// TIA Portal V16 export
// export: Created 2022-11-17T15:49:15.2421619Z, ExportSetting WithDefaults, DisplayName Totally Integrated Automation Portal, DisplayVersion V16 Update 6, DisplayName TIA Portal Version Control Interface, DisplayVersion V16 Update 2, DisplayName TIA Portal Openness, DisplayVersion V16 Update 6, DisplayName SINAMICS Startdrive Advanced, DisplayVersion V16 Update 5, DisplayName SINAMICS Startdrive G130, G150, S120, S150, SINAMICS MV, S210, DisplayVersion V16 Update 5, DisplayName SINAMICS Startdrive G110M, G120, G120C, G120D, G120P, G115D, DisplayVersion V16 Update 5, DisplayName STEP 7 Professional, DisplayVersion V16 Update 6, DisplayName STEP 7 Safety, DisplayVersion V16, DisplayName WinCC Advanced, DisplayVersion V16 Update 6
FUNCTION "FC06_TechnoplatCycle" : Void   // FC6, LAD
TITLE = Machine cycle
{ S7_Optimized_Access := 'FALSE' }
AUTHOR : Robopac
VERSION : 0.0
// stored: AutoNumber false, IsIECCheckEnabled false, SetENOAutomatically false, UDAEnableTagReadback false
   VAR_TEMP   // added for the SCL form of the ladder/FBD networks
      _w1 : Bool;
   END_VAR
BEGIN

REGION Network 1: Machine cycle: M0.0 Start cycle
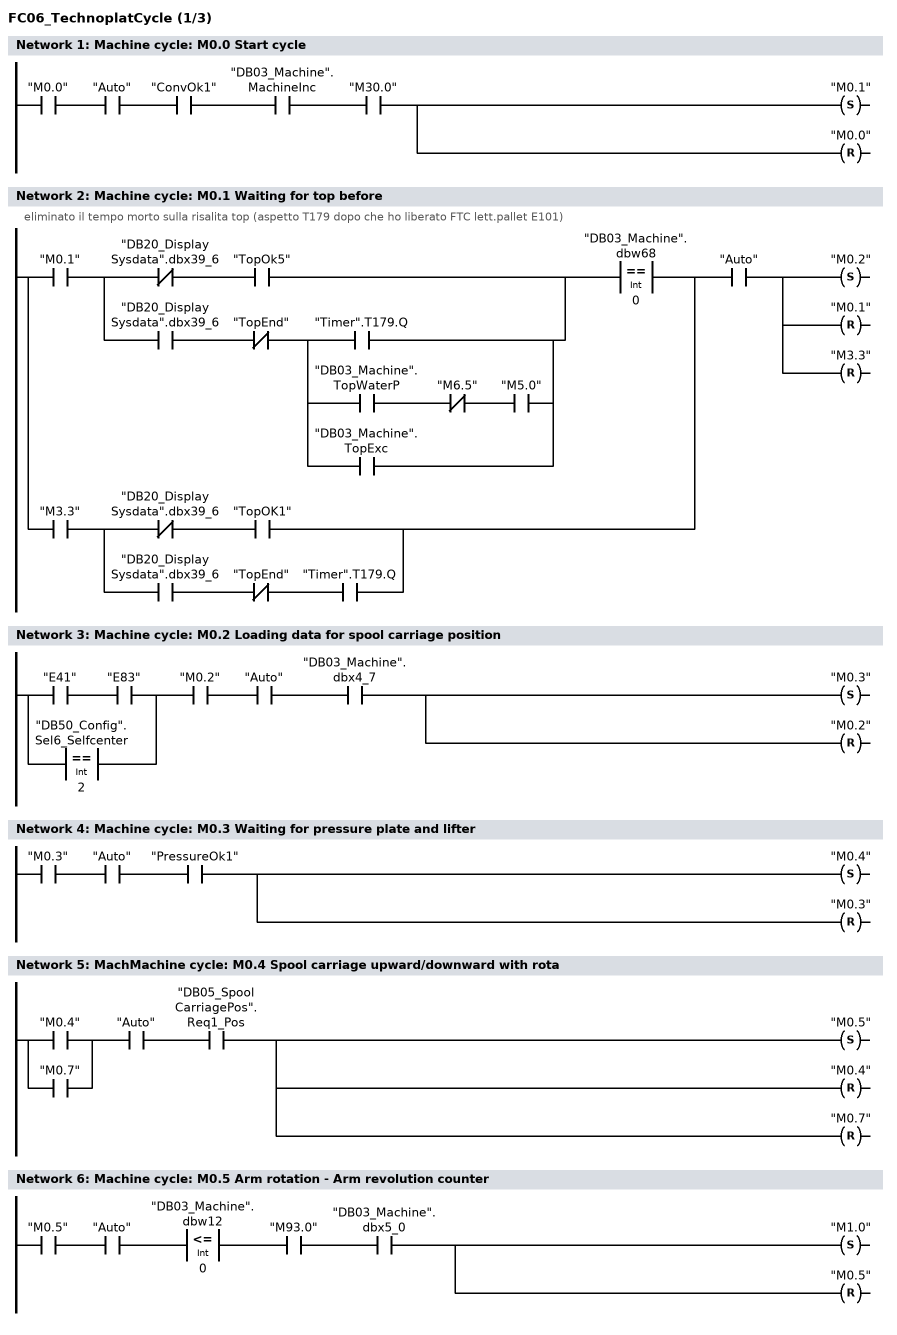
   RUNG wire#powerrail
      Contact( "M0.0" )
      Contact( "Auto" )
      Contact( "ConvOk1" )
      Contact( "DB03_Machine".MachineInc )
      Contact( "M30.0" )
      wire#w1
      S_Coil( "M0.1" )
   END_RUNG
   RUNG wire#w1
      R_Coil( "M0.0" )
   END_RUNG
   // the same network as SCL:
   IF "M0.0" AND "Auto" AND "ConvOk1" AND "DB03_Machine".MachineInc AND "M30.0" THEN
       "M0.1" := TRUE;
       "M0.0" := FALSE;
   END_IF;
END_REGION

REGION Network 2: Machine cycle: M0.1 Waiting for top before
   // eliminato il tempo morto sulla risalita top (aspetto T179 dopo che ho liberato FTC lett.pallet E101)
   RUNG wire#powerrail
      Contact( "M0.1" )
      wire#w1
      I_Contact( "DB20_DisplaySysdata".dbx39_6 )
      Contact( "TopOk5" )
      wire#w2
      { S7_Templates := "SrcType := Int" } EQ_Contact(in1 := "DB03_Machine".dbw68, in2 := 0)
      wire#w4
      Contact( "Auto" )
      wire#w6
      S_Coil( "M0.2" )
   END_RUNG
   RUNG wire#w1
      Contact( "DB20_DisplaySysdata".dbx39_6 )
      I_Contact( "TopEnd" )
      wire#w3
      Contact( "Timer".T179.Q )
   END_RUNG wire#w2
   RUNG wire#w3
      Contact( "DB03_Machine".TopWaterP )
      I_Contact( "M6.5" )
      Contact( "M5.0" )
   END_RUNG wire#w2
   RUNG wire#w3
      Contact( "DB03_Machine".TopExc )
   END_RUNG wire#w2
   RUNG wire#powerrail
      Contact( "M3.3" )
      wire#w5
      I_Contact( "DB20_DisplaySysdata".dbx39_6 )
      Contact( "TopOK1" )
   END_RUNG wire#w4
   RUNG wire#w5
      Contact( "DB20_DisplaySysdata".dbx39_6 )
      I_Contact( "TopEnd" )
      Contact( "Timer".T179.Q )
   END_RUNG wire#w4
   RUNG wire#w6
      R_Coil( "M0.1" )
   END_RUNG
   RUNG wire#w6
      R_Coil( "M3.3" )
   END_RUNG
   // the same network as SCL:
   IF (("M0.1" AND ((NOT "DB20_DisplaySysdata".dbx39_6 AND "TopOk5") OR ("DB20_DisplaySysdata".dbx39_6 AND NOT "TopEnd" AND ("Timer".T179.Q OR ("DB03_Machine".TopWaterP AND NOT "M6.5" AND "M5.0") OR "DB03_Machine".TopExc))) AND ("DB03_Machine".dbw68 = 0)) OR ("M3.3" AND ((NOT "DB20_DisplaySysdata".dbx39_6 AND "TopOK1") OR ("DB20_DisplaySysdata".dbx39_6 AND NOT "TopEnd" AND "Timer".T179.Q)))) AND "Auto" THEN
       "M0.2" := TRUE;
   END_IF;
   #_w1 := (("M0.1" AND ((NOT "DB20_DisplaySysdata".dbx39_6 AND "TopOk5") OR ("DB20_DisplaySysdata".dbx39_6 AND NOT "TopEnd" AND ("Timer".T179.Q OR ("DB03_Machine".TopWaterP AND NOT "M6.5" AND "M5.0") OR "DB03_Machine".TopExc))) AND ("DB03_Machine".dbw68 = 0)) OR ("M3.3" AND ((NOT "DB20_DisplaySysdata".dbx39_6 AND "TopOK1") OR ("DB20_DisplaySysdata".dbx39_6 AND NOT "TopEnd" AND "Timer".T179.Q)))) AND "Auto";
   IF #_w1 THEN
       "M0.1" := FALSE;
       "M3.3" := FALSE;
   END_IF;
END_REGION

REGION Network 3: Machine cycle: M0.2 Loading data for spool carriage position
   RUNG wire#powerrail
      Contact( "E41" )
      Contact( "E83" )
      wire#w1
      Contact( "M0.2" )
      Contact( "Auto" )
      Contact( "DB03_Machine".dbx4_7 )
      wire#w2
      S_Coil( "M0.3" )
   END_RUNG
   RUNG wire#powerrail
      { S7_Templates := "SrcType := Int" } EQ_Contact(in1 := "DB50_Config".Sel6_Selfcenter, in2 := 2)
   END_RUNG wire#w1
   RUNG wire#w2
      R_Coil( "M0.2" )
   END_RUNG
   // the same network as SCL:
   IF (("E41" AND "E83") OR ("DB50_Config".Sel6_Selfcenter = 2)) AND "M0.2" AND "Auto" AND "DB03_Machine".dbx4_7 THEN
       "M0.3" := TRUE;
       "M0.2" := FALSE;
   END_IF;
END_REGION

REGION Network 4: Machine cycle: M0.3 Waiting for pressure plate and lifter
   RUNG wire#powerrail
      Contact( "M0.3" )
      Contact( "Auto" )
      Contact( "PressureOk1" )
      wire#w1
      S_Coil( "M0.4" )
   END_RUNG
   RUNG wire#w1
      R_Coil( "M0.3" )
   END_RUNG
   // the same network as SCL:
   IF "M0.3" AND "Auto" AND "PressureOk1" THEN
       "M0.4" := TRUE;
       "M0.3" := FALSE;
   END_IF;
END_REGION

REGION Network 5: MachMachine cycle: M0.4 Spool carriage upward/downward with rota
   RUNG wire#powerrail
      Contact( "M0.4" )
      wire#w1
      Contact( "Auto" )
      Contact( "DB05_SpoolCarriagePos".Req1_Pos )
      wire#w2
      S_Coil( "M0.5" )
   END_RUNG
   RUNG wire#powerrail
      Contact( "M0.7" )
   END_RUNG wire#w1
   RUNG wire#w2
      R_Coil( "M0.4" )
   END_RUNG
   RUNG wire#w2
      R_Coil( "M0.7" )
   END_RUNG
   // the same network as SCL:
   IF ("M0.4" OR "M0.7") AND "Auto" AND "DB05_SpoolCarriagePos".Req1_Pos THEN "M0.5" := TRUE; END_IF;
   #_w1 := ("M0.4" OR "M0.7") AND "Auto" AND "DB05_SpoolCarriagePos".Req1_Pos;
   IF #_w1 THEN
       "M0.4" := FALSE;
       "M0.7" := FALSE;
   END_IF;
END_REGION

REGION Network 6: Machine cycle: M0.5 Arm rotation - Arm revolution counter
   RUNG wire#powerrail
      Contact( "M0.5" )
      Contact( "Auto" )
      { S7_Templates := "SrcType := Int" } LE_Contact(in1 := "DB03_Machine".dbw12, in2 := 0)
      Contact( "M93.0" )
      Contact( "DB03_Machine".dbx5_0 )
      wire#w1
      S_Coil( "M1.0" )
   END_RUNG
   RUNG wire#w1
      R_Coil( "M0.5" )
   END_RUNG
   // the same network as SCL:
   IF "M0.5" AND "Auto" AND ("DB03_Machine".dbw12 <= 0) AND "M93.0" AND "DB03_Machine".dbx5_0 THEN
       "M1.0" := TRUE;
       "M0.5" := FALSE;
   END_IF;
END_REGION

REGION Network 7: Machine cycle: M1.0 Revolution over welder contrast
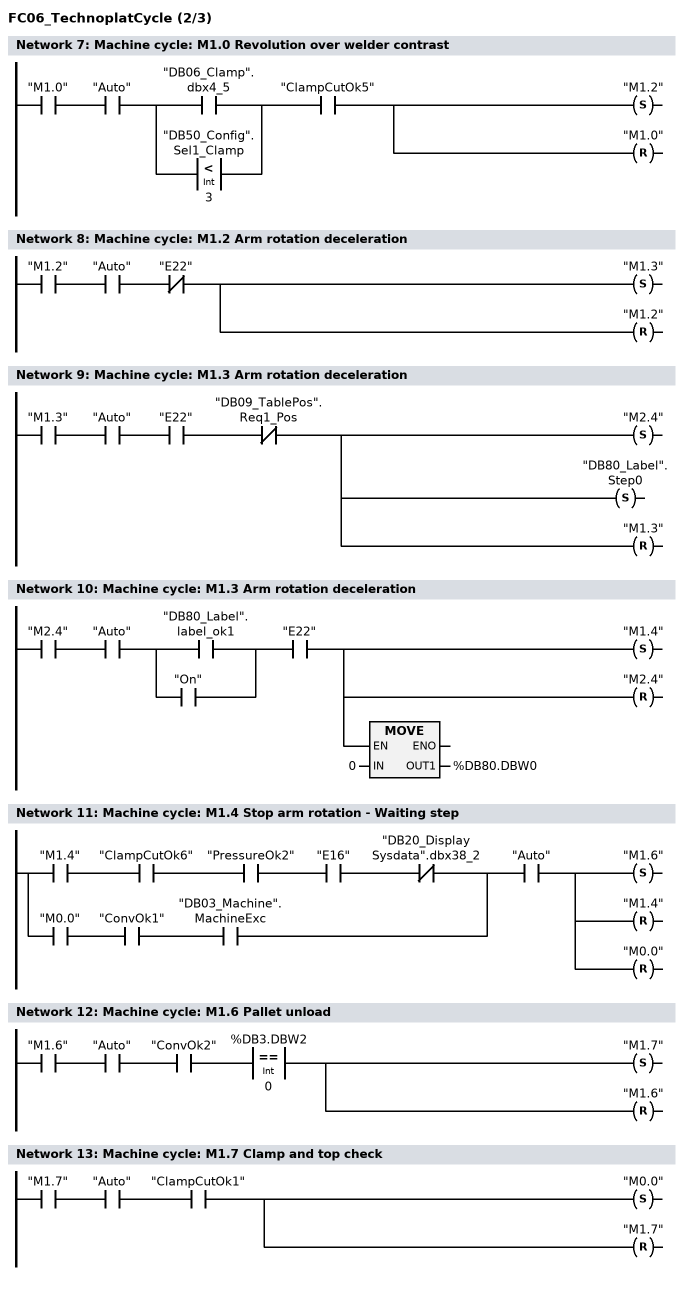
   RUNG wire#powerrail
      Contact( "M1.0" )
      Contact( "Auto" )
      wire#w1
      Contact( "DB06_Clamp".dbx4_5 )
      wire#w2
      Contact( "ClampCutOk5" )
      wire#w3
      S_Coil( "M1.2" )
   END_RUNG
   RUNG wire#w1
      { S7_Templates := "SrcType := Int" } LT_Contact(in1 := "DB50_Config".Sel1_Clamp, in2 := 3)
   END_RUNG wire#w2
   RUNG wire#w3
      R_Coil( "M1.0" )
   END_RUNG
   // the same network as SCL:
   IF "M1.0" AND "Auto" AND ("DB06_Clamp".dbx4_5 OR ("DB50_Config".Sel1_Clamp < 3)) AND "ClampCutOk5" THEN
       "M1.2" := TRUE;
       "M1.0" := FALSE;
   END_IF;
END_REGION

REGION Network 8: Machine cycle: M1.2 Arm rotation deceleration
   RUNG wire#powerrail
      Contact( "M1.2" )
      Contact( "Auto" )
      I_Contact( "E22" )
      wire#w1
      S_Coil( "M1.3" )
   END_RUNG
   RUNG wire#w1
      R_Coil( "M1.2" )
   END_RUNG
   // the same network as SCL:
   IF "M1.2" AND "Auto" AND NOT "E22" THEN
       "M1.3" := TRUE;
       "M1.2" := FALSE;
   END_IF;
END_REGION

REGION Network 9: Machine cycle: M1.3 Arm rotation deceleration
   RUNG wire#powerrail
      Contact( "M1.3" )
      Contact( "Auto" )
      Contact( "E22" )
      I_Contact( "DB09_TablePos".Req1_Pos )
      wire#w1
      S_Coil( "M2.4" )
   END_RUNG
   RUNG wire#w1
      S_Coil( "DB80_Label".Step0 )
   END_RUNG
   RUNG wire#w1
      R_Coil( "M1.3" )
   END_RUNG
   // the same network as SCL:
   IF "M1.3" AND "Auto" AND "E22" AND NOT "DB09_TablePos".Req1_Pos THEN
       "M2.4" := TRUE;
       "DB80_Label".Step0 := TRUE;
       "M1.3" := FALSE;
   END_IF;
END_REGION

REGION Network 10: Machine cycle: M1.3 Arm rotation deceleration
   RUNG wire#powerrail
      Contact( "M2.4" )
      Contact( "Auto" )
      wire#w1
      Contact( "DB80_Label".label_ok1 )
      wire#w2
      Contact( "E22" )
      wire#w3
      S_Coil( "M1.4" )
   END_RUNG
   RUNG wire#w1
      Contact( "On" )
   END_RUNG wire#w2
   RUNG wire#w3
      R_Coil( "M2.4" )
   END_RUNG
   RUNG wire#w3
      { S7_GenerateENO := "TRUE" } Move(in := 0, out1 => %DB80.DBW0)
   END_RUNG
   // the same network as SCL:
   IF "M2.4" AND "Auto" AND ("DB80_Label".label_ok1 OR "On") AND "E22" THEN "M1.4" := TRUE; END_IF;
   #_w1 := "M2.4" AND "Auto" AND ("DB80_Label".label_ok1 OR "On") AND "E22";
   IF #_w1 THEN
       "M2.4" := FALSE;
       %DB80.DBW0 := 0;
   END_IF;
END_REGION

REGION Network 11: Machine cycle: M1.4 Stop arm rotation - Waiting step
   RUNG wire#powerrail
      Contact( "M1.4" )
      Contact( "ClampCutOk6" )
      Contact( "PressureOk2" )
      Contact( "E16" )
      I_Contact( "DB20_DisplaySysdata".dbx38_2 )
      wire#w1
      Contact( "Auto" )
      wire#w2
      S_Coil( "M1.6" )
   END_RUNG
   RUNG wire#powerrail
      Contact( "M0.0" )
      Contact( "ConvOk1" )
      Contact( "DB03_Machine".MachineExc )
   END_RUNG wire#w1
   RUNG wire#w2
      R_Coil( "M1.4" )
   END_RUNG
   RUNG wire#w2
      R_Coil( "M0.0" )
   END_RUNG
   // the same network as SCL:
   IF (("M1.4" AND "ClampCutOk6" AND "PressureOk2" AND "E16" AND NOT "DB20_DisplaySysdata".dbx38_2) OR ("M0.0" AND "ConvOk1" AND "DB03_Machine".MachineExc)) AND "Auto" THEN
       "M1.6" := TRUE;
   END_IF;
   #_w1 := (("M1.4" AND "ClampCutOk6" AND "PressureOk2" AND "E16" AND NOT "DB20_DisplaySysdata".dbx38_2) OR ("M0.0" AND "ConvOk1" AND "DB03_Machine".MachineExc)) AND "Auto";
   IF #_w1 THEN
       "M1.4" := FALSE;
       "M0.0" := FALSE;
   END_IF;
END_REGION

REGION Network 12: Machine cycle: M1.6 Pallet unload
   RUNG wire#powerrail
      Contact( "M1.6" )
      Contact( "Auto" )
      Contact( "ConvOk2" )
      { S7_Templates := "SrcType := Int" } EQ_Contact(in1 := %DB3.DBW2, in2 := 0)
      wire#w1
      S_Coil( "M1.7" )
   END_RUNG
   RUNG wire#w1
      R_Coil( "M1.6" )
   END_RUNG
   // the same network as SCL:
   IF "M1.6" AND "Auto" AND "ConvOk2" AND (%DB3.DBW2 = 0) THEN
       "M1.7" := TRUE;
       "M1.6" := FALSE;
   END_IF;
END_REGION

REGION Network 13: Machine cycle: M1.7 Clamp and top check
   RUNG wire#powerrail
      Contact( "M1.7" )
      Contact( "Auto" )
      Contact( "ClampCutOk1" )
      wire#w1
      S_Coil( "M0.0" )
   END_RUNG
   RUNG wire#w1
      R_Coil( "M1.7" )
   END_RUNG
   // the same network as SCL:
   IF "M1.7" AND "Auto" AND "ClampCutOk1" THEN
       "M0.0" := TRUE;
       "M1.7" := FALSE;
   END_IF;
END_REGION

REGION Network 14: Machine cycle: M0.5 Arm rotation - Arm revolution counter
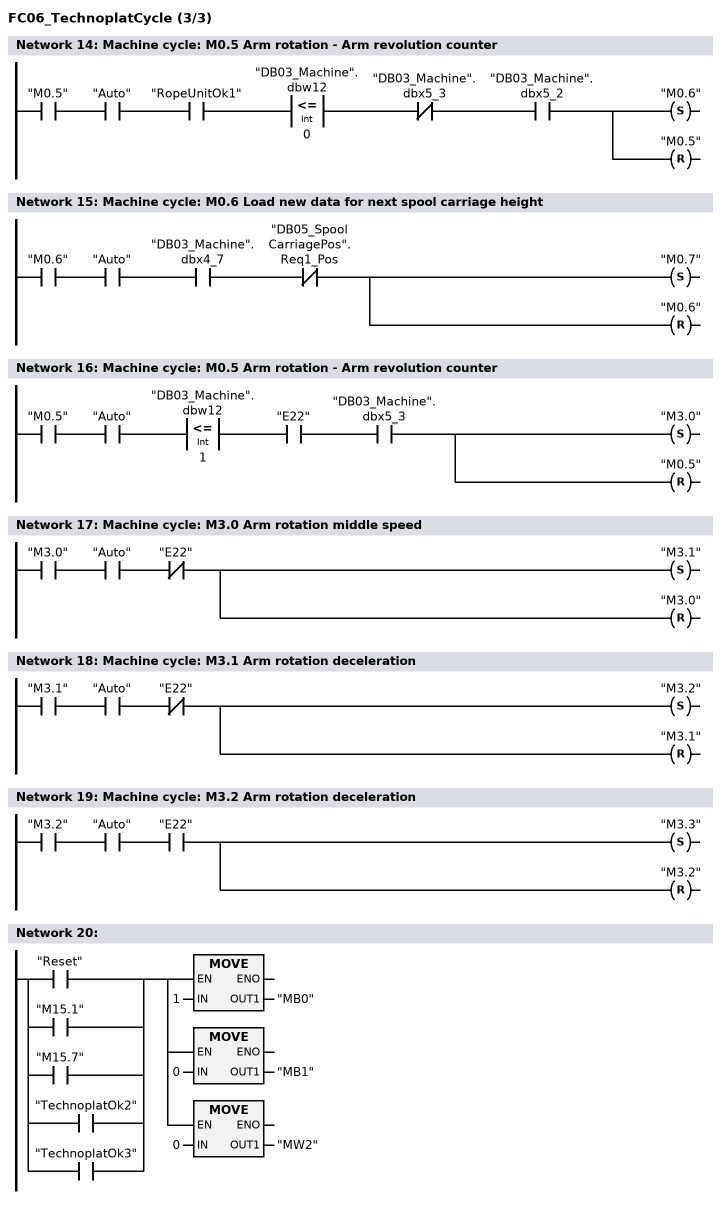
   RUNG wire#powerrail
      Contact( "M0.5" )
      Contact( "Auto" )
      Contact( "RopeUnitOk1" )
      { S7_Templates := "SrcType := Int" } LE_Contact(in1 := "DB03_Machine".dbw12, in2 := 0)
      I_Contact( "DB03_Machine".dbx5_3 )
      Contact( "DB03_Machine".dbx5_2 )
      wire#w1
      S_Coil( "M0.6" )
   END_RUNG
   RUNG wire#w1
      R_Coil( "M0.5" )
   END_RUNG
   // the same network as SCL:
   IF "M0.5" AND "Auto" AND "RopeUnitOk1" AND ("DB03_Machine".dbw12 <= 0) AND NOT "DB03_Machine".dbx5_3 AND "DB03_Machine".dbx5_2 THEN
       "M0.6" := TRUE;
       "M0.5" := FALSE;
   END_IF;
END_REGION

REGION Network 15: Machine cycle: M0.6 Load new data for next spool carriage height
   RUNG wire#powerrail
      Contact( "M0.6" )
      Contact( "Auto" )
      Contact( "DB03_Machine".dbx4_7 )
      I_Contact( "DB05_SpoolCarriagePos".Req1_Pos )
      wire#w1
      S_Coil( "M0.7" )
   END_RUNG
   RUNG wire#w1
      R_Coil( "M0.6" )
   END_RUNG
   // the same network as SCL:
   IF "M0.6" AND "Auto" AND "DB03_Machine".dbx4_7 AND NOT "DB05_SpoolCarriagePos".Req1_Pos THEN
       "M0.7" := TRUE;
       "M0.6" := FALSE;
   END_IF;
END_REGION

REGION Network 16: Machine cycle: M0.5 Arm rotation - Arm revolution counter
   RUNG wire#powerrail
      Contact( "M0.5" )
      Contact( "Auto" )
      { S7_Templates := "SrcType := Int" } LE_Contact(in1 := "DB03_Machine".dbw12, in2 := 1)
      Contact( "E22" )
      Contact( "DB03_Machine".dbx5_3 )
      wire#w1
      S_Coil( "M3.0" )
   END_RUNG
   RUNG wire#w1
      R_Coil( "M0.5" )
   END_RUNG
   // the same network as SCL:
   IF "M0.5" AND "Auto" AND ("DB03_Machine".dbw12 <= 1) AND "E22" AND "DB03_Machine".dbx5_3 THEN
       "M3.0" := TRUE;
       "M0.5" := FALSE;
   END_IF;
END_REGION

REGION Network 17: Machine cycle: M3.0 Arm rotation middle speed
   RUNG wire#powerrail
      Contact( "M3.0" )
      Contact( "Auto" )
      I_Contact( "E22" )
      wire#w1
      S_Coil( "M3.1" )
   END_RUNG
   RUNG wire#w1
      R_Coil( "M3.0" )
   END_RUNG
   // the same network as SCL:
   IF "M3.0" AND "Auto" AND NOT "E22" THEN
       "M3.1" := TRUE;
       "M3.0" := FALSE;
   END_IF;
END_REGION

REGION Network 18: Machine cycle: M3.1 Arm rotation deceleration
   RUNG wire#powerrail
      Contact( "M3.1" )
      Contact( "Auto" )
      I_Contact( "E22" )
      wire#w1
      S_Coil( "M3.2" )
   END_RUNG
   RUNG wire#w1
      R_Coil( "M3.1" )
   END_RUNG
   // the same network as SCL:
   IF "M3.1" AND "Auto" AND NOT "E22" THEN
       "M3.2" := TRUE;
       "M3.1" := FALSE;
   END_IF;
END_REGION

REGION Network 19: Machine cycle: M3.2 Arm rotation deceleration
   RUNG wire#powerrail
      Contact( "M3.2" )
      Contact( "Auto" )
      Contact( "E22" )
      wire#w1
      S_Coil( "M3.3" )
   END_RUNG
   RUNG wire#w1
      R_Coil( "M3.2" )
   END_RUNG
   // the same network as SCL:
   IF "M3.2" AND "Auto" AND "E22" THEN
       "M3.3" := TRUE;
       "M3.2" := FALSE;
   END_IF;
END_REGION

REGION Network 20
   RUNG wire#powerrail
      Contact( "Reset" )
      wire#w1
      { S7_GenerateENO := "TRUE" } Move(in := 1, out1 => "MB0")
   END_RUNG
   RUNG wire#powerrail
      Contact( "M15.1" )
   END_RUNG wire#w1
   RUNG wire#powerrail
      Contact( "M15.7" )
   END_RUNG wire#w1
   RUNG wire#powerrail
      Contact( "TechnoplatOk2" )
   END_RUNG wire#w1
   RUNG wire#powerrail
      Contact( "TechnoplatOk3" )
   END_RUNG wire#w1
   RUNG wire#w1
      { S7_GenerateENO := "TRUE" } Move(in := 0, out1 => "MB1")
   END_RUNG
   RUNG wire#w1
      { S7_GenerateENO := "TRUE" } Move(in := 0, out1 => "MW2")
   END_RUNG
   // the same network as SCL:
   IF "Reset" OR "M15.1" OR "M15.7" OR "TechnoplatOk2" OR "TechnoplatOk3" THEN
       "MB0" := 1;
       "MB1" := 0;
       "MW2" := 0;
   END_IF;
END_REGION
END_FUNCTION
